PROGRAM MAIN
VAR
END_VAR

END_PROGRAM

(* stored: Version 1.1.0.1
   POU MAIN: Id {c2dc4aad-864e-432c-a950-ffd3625488fc} *)
